Yaskawa INFORM job: _DEL19.JBI

/JOB
//NAME _DEL19
//POS
///NPOS 0,0,0,0,0,0
//INST
///DATE 2018/08/30 09:53
///ATTR SC,RW,SY
///GROUP1 ST1
NOP
END
